// TIA Portal V20 export
TYPE "typeCmControlNodeSoftCam"
// stored: Namespace Unit1.Em13
   STRUCT
      jrUnIoadingPnPAxisX : "Unit1.Em13.typeCmControlNodeSoftCamjrUnIoadingPnPAxisX";
      jrUnIoadingPnPAxisZ : "Unit1.Em13.typeCmControlNodeSoftCamjrUnIoadingPnPAxisZ";
      jrUnIoadingPnPAxisC : "Unit1.Em13.typeCmControlNodeSoftCamjrUnIoadingPnPAxisC";
   END_STRUCT;
END_TYPE
